ADAPTER Callback (* Message Callback *)
  (* Standard: 61499-1 *)
  (* Version 1.0, 2025-09-06, Franz Höpfinger *)
  PACKAGE isobus::pgn::tx;
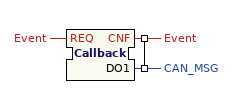
  EVENT_INPUT
    REQ; (* Request from Socket *)
  END_EVENT
  EVENT_OUTPUT
    CNF WITH DO1; (* Confirmation from Plug *)
  END_EVENT
  VAR_OUTPUT
    DO1 : isobus::pgn::CAN_MSG;
  END_VAR
END_ADAPTER
